PROGRAM PR_Conveyor_Out
VAR
	fSpeed_Conveyor			: REAL := 25;
	bUp_Speed				: BOOL;
	bDw_Speed				: BOOL;
	bMotor_Conveyor			: BOOL;
	fb_Conveyor				: FB_FoodMixerModule;
END_VAR

fb_Conveyor(nLine:= 3, UnitID:= 3, fSpeed_motor_mixer:= fSpeed_Conveyor);

ACTION Auto:
fb_Conveyor.Auto();
END_ACTION

ACTION Manual:
fb_Conveyor.Manual(bUp_Motor_Mixer := bUp_Speed, bDown_Motor_Mixer := bDw_Speed,
					bMotor_mixer_Manual := bMotor_Conveyor,bMotor_mixer_reverse := FALSE);
IF bUp_Speed THEN
	bUp_Speed := FALSE;
END_IF

IF bDw_Speed THEN
	bDw_Speed := FALSE;
END_IF
END_ACTION

ACTION Reset:
fb_Conveyor.Reset();
END_ACTION

ACTION Stop:
bMotor_Conveyor		:= FALSE;
fb_Conveyor.Stop();
END_ACTION

END_PROGRAM

(* stored: Version 1.1.0.1, ProductVersion 3.1.4024.12
   POU PR_Conveyor_Out: Id {8c087792-927f-4f94-8161-60b452cc5a6e}, SpecialFunc None
   Action Auto: Id {6fceea7e-2008-4adf-8698-130b8460b778}
   Action Manual: Id {e931e9fb-a624-483c-b894-cabc04e96d69}
   Action Reset: Id {a9385318-48d6-4b78-875d-9ffa56d20e30}
   Action Stop: Id {3d1ea182-ce8d-4f25-86c5-57cd8aa01916} *)
